// TIA Portal project "Forward_and_Reserve_Operation_3-Phase_Motor" (V15)
// FORWARD AND REVERSE OPERATION OF A 3-PHASE MOTOR

(* hardware
DEVICE "S7-1200 station_1"  S7-1200 Station
   slot 0: "Rack_0"  S7-1200 Rack  Rack  V1.0
   slot 1: "PLC_1"  CPU 1212C DC/DC/DC  6ES7 212-1AE40-0XB0  V4.2
*)

// ===== PLC "PLC_1"  CPU 1212C DC/DC/DC =====

VAR_GLOBAL   // PLC tag table "Default tag table"
   "I_THERMAL_RELAY" AT %I0.0 : Bool;
   "I_START_BTN_1" AT %I0.1 : Bool;
   "I_STOP_BTN" AT %I0.2 : Bool;
   "I_FOWARD_BTN" AT %I0.3 : Bool;
   "I_RESERVE_BTN" AT %I0.4 : Bool;
   "Q_FOWARD_MOTOR" AT %Q0.0 : Bool;
   "Q_RESERVE_MOTOR" AT %Q0.1 : Bool;
   "I_START_BTN_2" AT %I0.5 : Bool;
END_VAR

ORGANIZATION_BLOCK "Main"   // OB1, LAD, ProgramCycle
TITLE = "Main Program Sweep (Cycle)"
{ S7_Optimized_Access := 'TRUE' }
VERSION : 0.1
   VAR_INPUT
      Initial_Call : Bool;   // Initial call of this OB
      Remanence : Bool;   // =True, if remanent data are available
   END_VAR
BEGIN

REGION Network 1: FORWARD
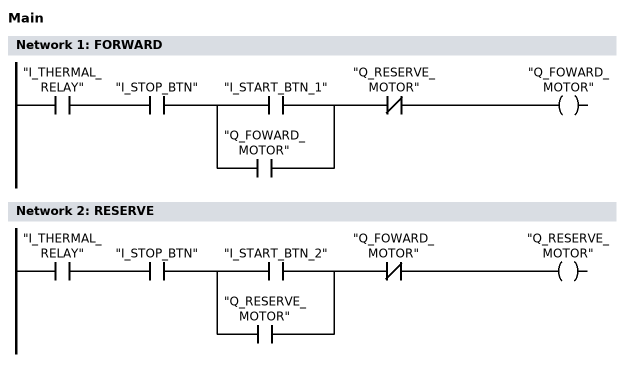
   RUNG wire#powerrail
      Contact( "I_THERMAL_RELAY" )
      Contact( "I_STOP_BTN" )
      wire#w1
      Contact( "I_START_BTN_1" )
      wire#w2
      I_Contact( "Q_RESERVE_MOTOR" )
      Coil( "Q_FOWARD_MOTOR" )
   END_RUNG
   RUNG wire#w1
      Contact( "Q_FOWARD_MOTOR" )
   END_RUNG wire#w2
   // the same network as SCL:
   "Q_FOWARD_MOTOR" := "I_THERMAL_RELAY" AND "I_STOP_BTN" AND ("I_START_BTN_1" OR "Q_FOWARD_MOTOR") AND NOT "Q_RESERVE_MOTOR";
END_REGION

REGION Network 2: RESERVE
   RUNG wire#powerrail
      Contact( "I_THERMAL_RELAY" )
      Contact( "I_STOP_BTN" )
      wire#w1
      Contact( "I_START_BTN_2" )
      wire#w2
      I_Contact( "Q_FOWARD_MOTOR" )
      Coil( "Q_RESERVE_MOTOR" )
   END_RUNG
   RUNG wire#w1
      Contact( "Q_RESERVE_MOTOR" )
   END_RUNG wire#w2
   // the same network as SCL:
   "Q_RESERVE_MOTOR" := "I_THERMAL_RELAY" AND "I_STOP_BTN" AND ("I_START_BTN_2" OR "Q_RESERVE_MOTOR") AND NOT "Q_FOWARD_MOTOR";
END_REGION
END_ORGANIZATION_BLOCK